INTERFACE I_AuditLogListener

METHOD OnTraceReceived
VAR_INPUT
    message : ST_AuditLogMessages;
END_VAR
END_METHOD

END_INTERFACE

(* stored: Version 1.1.0.1
   Itf I_AuditLogListener: Id {04bb2395-4105-409e-ab3b-a8e8b2124287}
   Method OnTraceReceived: Id {a4e1ddd1-aea8-4100-9520-2052d32fc5cf} *)
